(* CoDeSys 2.3.9.62 project: PackML_StateModel_Example_v2-3.pro *)
(* Libraries: STANDARD.LIB 5.6.98 13:03:02 *)

(* Global variable list: Global_Variables *)
VAR_GLOBAL
(* -------------INPUTS-------------------*)
	I_Btn_Reset			(*AT %I* *)		:BOOL;	(*Reset button*)
	I_Btn_Start			(* AT %I* *)	:BOOL;	(*Start button*)
	I_Btn_Stop			(* AT %I* *)	:BOOL;	(*Stop button*)
	I_EStopClear 		(* AT %I* *)	:BOOL :=TRUE;	(*EStop is cleared*)
	I_CoversClosed 		(* AT %I* *)	:BOOL :=TRUE;	(*Covers are completely closed*)

(* -------------OUTPUTS-------------------*)
	O_LightON_up 		(* AT %Q* *)	:BOOL;	(*Light ON - Up*)
	O_LightON_low 		(* AT %Q* *)	:BOOL;	(*Light ON - Lower*)
	OuLight_up 			(* AT %Q* *)	:INT;	(*Light Analog - Up*)
	OuLight_low 		(* AT %Q* *)	:INT;	(*Light Analog - Lower*)
	O_Light_Start 		(* AT %Q* *)	:BOOL;	(*Light Button Start*)
	O_Light_Stop 		(* AT %Q* *)	:BOOL;	(*Light Button Stop*)
	O_Light_Warning 		(* AT %Q* *):BOOL;	(*Light Button Warning*)
	O_Light_Error 		(* AT %Q* *)	:BOOL;	(*Light Button Error*)
	O_RelayStop 			(* AT %Q* *):BOOL;	(*Relay out : Stop*)
	O_RelayEStop			(* AT %Q* *):BOOL;	(*Relay out : EStop*)
	O_RelayEnableLED_Pwr_Along	(* AT %Q* *):BOOL;	(*Relay out : Enable LED power along belt*)

	bReset_System		: BOOL;			(*System reset*)
	bReset_System_Long	: BOOL;			(*System reset - Long*)
	bReqShutdown		: BOOL;			(*Request shutdown*)
	bDisplayOn			: BOOL;			(*Display on*)

(* -------------HMI INPUTS (from HMI to PLC) -------------------*)
	HMI_wControlWord	: WORD;			(*Control bits: 0=*)
	HMI_uModeReq		: UINT :=5;		(*Mode request. DEFAULT:PRODUCTION1*)

(* -------------HMI OUTPUTS (from PLC to HMI) -------------------*)
	PLC_wStatusWord		: WORD;			(*Status bits: 0=*)
	PLC_uModeCurrent	: UINT;			(*Current Mode*)
	PLC_uStateCurrent	: UINT;			(*Current State*)
	fAngle1				: REAL := 50;	(*Process: Angle1*)
	fAngle2				: REAL := 90;	(*Process: Angle2*)


(*-----------------------FUNCTION BLOCKS----------------*)
	fbStateModel		: FB_PackMLStateModel_ST;	(*FB for executing PackML state model*)

(*-----------------------OTHER GLOBAL VARS ----------------*)
	uCounterPosCurr_SIMU	: UDINT;	(*Current Counter position*)

END_VAR

(*------------------------- PERSISTENT VARIABLES --------------------------------*)
VAR_GLOBAL PERSISTENT

END_VAR

(*------------------------- CONSTANT VARIABLES --------------------------------*)
VAR_GLOBAL CONSTANT
(*-----------------------Setup Constants----------------------------*)
	bSIMU			: BOOL 	:= TRUE;	(*In simulation mode*)

(*-----------------------TIME Constants----------------------------*)
	TRESET_SYSTEM	: TIME := T#3s;		(*Delay for System Reset*)
	TRESET_LONG		: TIME := T#10s;	(*Delay for Long Reset*)

END_VAR

(* Data type *)
TYPE E_Mode :
(*UserModes: Modes for different production states*)
(
	eMode_undefined := 0,
	eMode_Automatic :=1,
	eMode_Manual :=3,
	eMode_Production1 :=5,
	eMode_Production2 :=6
);
END_TYPE

(* Data type *)
TYPE E_ModeProc :
(*Procedural control modes. Can be changed in any state*)
(
	eModeProc_undefined := 0,
	eModeProc_Automatic :=1,
	eModeProc_SemiAutomatic :=2,
	eModeProc_Manual :=3
);
END_TYPE

(* Data type *)
TYPE E_PackMLState :
(*PackML States*)
(
	eSt_Aborting :=0,
	eSt_Aborted,
	eSt_Clearing,
	eSt_Stopped,
	eSt_Stopping,
	eSt_Resetting,
	eSt_Idle,
	eSt_Starting,
	eSt_Execute,
	eSt_Suspending,
	eSt_Suspended,
	eSt_Unsuspending,
	eSt_Holding,
	eSt_Held,
	eSt_UnHolding,
	eSt_Completing,
	eSt_Completed
);
END_TYPE

(* POU Programs/PRG_Application, ST *)
PROGRAM PRG_Application
VAR
	bInitDone	: BOOL;
END_VAR
(*Application specific program routine.*)
(* It can utilise the same main state model and modes also internally, and filtter
its execution conditions according that information. Alternative option is to call
this program from Main, but only when certain conditions are met. Then special care 
should be taken what the outputs are when it is NOT called!.*)


(*Initialisation procedures*)
IF NOT bInitDone THEN
	(*TODO: Do some init actions*)
	bInitDone:=TRUE;
END_IF;

(*Mode and state analysis*)
(*Execution mode*)
IF bSIMU THEN
	PRG_SIMU();
END_IF;


IF (fbStateModel.eState >= eSt_Stopped) THEN
	(*State is equal or above Stopped*)			(*TODO: Remove/Replace this row with desired actions*)
	CASE fbStateModel.eMode OF
		(*MODE: MANUAL*)
		eMode_Manual:
			(*TODO: Do some actions in manual mode*)
			(*E.g. calling some other PRG or FB implementing manual operations*)
			;									(*TODO: Remove/Replace this row with desired actions*)

		(*MODE: AUTOMATIC*)
		eMode_Automatic:
			(*TODO: Do some actions in automatic mode*)
			(*E.g. calling some other PRG or FB implementing automatic operations*)
			;									(*TODO: Remove/Replace this row with desired actions*)
		ELSE	(*Error*)
			; (*TODO*)
	END_CASE;
END_IF;


(*Enable LED powers*)
O_RelayEnableLED_Pwr_Along := (fbStateModel.eState >= eSt_Stopped);	(*TODO: Remove/Replace this row with desired actions*)


(*Clear LED output values in case 'low' states *)
IF (fbStateModel.eState <= eSt_Clearing) THEN
	(*TODO: Actions for clearing states *)
	(*UP*)
	O_LightON_up := FALSE;				(*TODO: Remove/Replace this row with desired actions*)
	OuLight_up := 0;					(*TODO: Change...*)
	(*Low*)
	O_LightON_low := FALSE;				(*TODO: Change...*)
	OuLight_low := 0;
END_IF;
END_PROGRAM

(* POU Programs/PRG_SIMU, ST *)
PROGRAM PRG_SIMU
VAR
	c	: INT;
END_VAR
(*This just simulator part, when program is used in simulated environment*)
IF fbStateModel.eState = eSt_Clearing THEN
uCounterPosCurr_SIMU := 0;
END_IF;

IF (fbStateModel.eState > eSt_Idle) AND (fbStateModel.eState < eSt_Completed) AND
		NOT ((fbStateModel.eState = eSt_Held) OR (fbStateModel.eState = eSt_Suspended)) THEN
	c:=c+1;
	IF c >= 5 THEN
		uCounterPosCurr_SIMU := uCounterPosCurr_SIMU + 1;
		c:=0;
	END_IF;
END_IF;
END_PROGRAM

(* POU Programs/PRG_Blinking, ST *)
PROGRAM PRG_Blinking
(*Avustavia laskentaoperaatioita
- vilkutussignaalit
Author: Niko Siltala, niko.siltala@tut.fi, Tampere University of Technology / MEI
Date: 2016-12-12
Version: 1.0
*)
VAR_OUTPUT
	bSign4Hz:BOOL;					(*4 Hz (240krt/min) taajudella vaihteleva signaali*)
	bSign2Hz:BOOL;					(*2 Hz (120krt/min) taajudella vaihteleva signaali*)
	bSign1Hz:BOOL;					(*1 Hz (60krt/min) taajudella vaihteleva signaali*)
	bSign0_5Hz:BOOL;				(*0,5 Hz (30krt/min) taajudella vaihteleva signaali*)
END_VAR
VAR
	bInitDone	: BOOL	:=FALSE;	(*Ohjelman initialisointi*)
	TP_Delay:TP;				(*Nopein taajuus / 2 tuottaja*)
	bBaseHz:BOOL:=FALSE;		(*Nopein taajuus/2*)
	iBaseHz:UINT:=4;				(*Base taajuus (Hz)*)
	(*RTRIG_BASE: R_TRIG;		(*Base signaali nousee*)*)
	RTRIG_2Hz_Sign : R_TRIG;		(*2Hz signaalin generointi*)
	RTRIG_1Hz_Sign : R_TRIG;		(*1Hz signaalin generointi*)
	RTRIG_0_5Hz_Sign : R_TRIG;	(*0,5Hz signaalin generointi*)
	tBaseTaajuus:TIME;			(*Base vilkutuksen timerin arvo. f/2*)
	fPLC_CYCLE_TIME: LREAL;	(*PLC:n cycli aika. Sekunttia*)

END_VAR
(*Ohjelman initialisoinnit - Suoritetaan vain kertaalleen*)
IF NOT bInitDone THEN
	(*fPLC_CYCLE_TIME := UDINT_TO_LREAL(SystemTaskInfoArr[1].cycleTime) / 10E6; (*[s]*)*)
	fPLC_Cycle_Time := 1;	(*[s]*)
	(*Base Vilkkusignaalien tuottaminen*)
	(* 250ms - 1* cykliaika(20ms)*)
	tBaseTaajuus := LREAL_TO_TIME( ( (1/ UINT_TO_LREAL(iBaseHz) / 2 ) - 1 * fPLC_CYCLE_TIME ) * 1000);
	bInitDone := TRUE;
END_IF;

(*Base signaalin genrointi*)
TP_Delay(IN:=NOT TP_Delay.Q , PT:=tBaseTaajuus);
IF NOT TP_Delay.Q THEN
	bBaseHz := NOT bBaseHz;
	bSign4Hz:= bBaseHz;
END_IF;

(*2Hz signaalin genrointi*)
RTRIG_2Hz_Sign(CLK:=bSign4Hz);
IF RTRIG_2Hz_Sign.Q THEN
	bSign2Hz:=NOT bSign2Hz;
END_IF;

(*1Hz signaalin genrointi*)
RTRIG_1Hz_Sign(CLK:=bSign2Hz);
IF RTRIG_1Hz_Sign.Q THEN
	bSign1Hz:=NOT bSign1Hz;
END_IF;

(*0,5 Hz signaalin generointi*)
RTRIG_0_5Hz_Sign(CLK:=bSign1Hz);
IF (RTRIG_0_5Hz_Sign.Q) THEN
	bSign0_5Hz:= NOT bSign0_5Hz;
END_IF;
END_PROGRAM

(* POU Programs/PRG_Initialisation, SFC *)
PROGRAM PRG_Initialisation
(*Example program to demonstrate imagenary Initialisation and Homing process*)
VAR_INPUT
	bReset		: BOOL;	(*Performs reset*)
END_VAR
VAR_OUTPUT
	bInitDone	: BOOL;	(*Initialisation is completed*)
END_VAR
VAR
	SFCReset 	: BOOL;	(*Resets the execution of SFC to init once this SFCFlag is set true *)
END_VAR
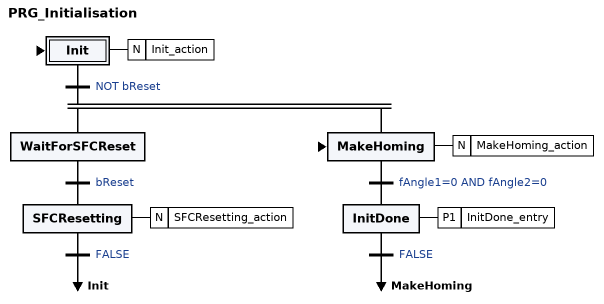
INITIAL_STEP Init:
	Init_action(N);
END_STEP
TRANSITION FROM Init TO (WaitForSFCReset, MakeHoming) := NOT bReset;
END_TRANSITION
STEP WaitForSFCReset:
END_STEP
TRANSITION FROM WaitForSFCReset TO SFCResetting := bReset;
END_TRANSITION
STEP SFCResetting:
	SFCResetting_action(N);
END_STEP
TRANSITION FROM SFCResetting TO Init := FALSE;
END_TRANSITION
STEP MakeHoming:
	MakeHoming_action(N);
END_STEP
TRANSITION FROM MakeHoming TO InitDone := fAngle1=0 AND fAngle2=0;
END_TRANSITION
STEP InitDone:
	InitDone_entry(P1);
END_STEP
TRANSITION FROM InitDone TO MakeHoming := FALSE;
END_TRANSITION

ACTION Init_action:
SFCReset := FALSE;
bReset	:= FALSE;
END_ACTION

ACTION SFCResetting_action:
SFCReset := TRUE;
END_ACTION

ACTION MakeHoming_action:
bInitDone := FALSE;
(*Return pointer1 to home. CCW rotation*)
fAngle1 := fAngle1 - 0.5;
IF fAngle1 <= 0 THEN
	fAngle1 := 0;
END_IF;

(*Return pointer2 to home. CCW rotation*)
IF fAngle2 <> 0 THEN
	IF fAngle2 < 0 THEN
		fAngle2 := fAngle2 + 360;
	END_IF;
	fAngle2 := fAngle2 - 0.5;
	IF fAngle2 <= 0 THEN
		fAngle2 := 0;
	END_IF;
END_IF;
END_ACTION

ACTION InitDone_entry:
bInitDone := TRUE;
END_ACTION
END_PROGRAM

(* POU PRG_MAIN, ST *)
PROGRAM PRG_MAIN
VAR
	TON_Reset_Long		: TON;
	TON_Reset_System	: TON;
	tonStarting			: TON;
	bBlink				: BOOL;	(*1s blinking for CodeSys Simulation*)
	c					: INT;	(*Support variable for blinking*)
	fbProcess3		: FB_Process3; (*FB Instance representing Process 3 *)
END_VAR
(* ****** Section 1: Initialisations and default values. Initial conditions for variables on every PLC cycle*)
fbStateModel.bSC := FALSE;
fbProcess3.packML_State := fbStateModel.eState;
fbProcess3.packML_Mode := fbStateModel.eMode;

PRG_MAIN_SAMPLE();

IF bSIMU THEN
	(*TODO set counter source*)
	;
END_IF;

(*System resets*)
TON_Reset_System(IN:=I_Btn_Reset,
		PT:=TRESET_SYSTEM ,
		Q=> , ET=> );		(*Simple Reset actions should happen after this*)
TON_Reset_Long(IN:=I_Btn_Reset,
		PT:=TRESET_LONG ,
		Q=>bReset_System_Long , ET=> );	(*Complete Reset actions should happen after this*)
bReset_System := TON_Reset_System.Q;

(* ****** Section 2: Grouping PackML states for calling Programs or FB instances.
This is to avoid repetition inside case structure in Section 3. With IF clause setting lower (and upper) state limits we can filter out the states when we want to call 
specific programs. The order of states is defined in Tab:Data types > E_PackMLState. eSt_Aborting is lowest and eSt_Completed is highest.
Here we filter calling programs, only when we are in higher states than Stopped. Inside IF there is again CASE which process each Control Mode separately.*)
(*Execution part. Making calls for program if we are on states above Stopped*)
IF (fbStateModel.eState > eSt_Stopped) THEN
	(*State is equal or above Stopped*)			(*TODO: Remove/Replace this row with desired actions*)
	CASE fbStateModel.eMode OF
		(*MODE: MANUAL*)
		eMode_Manual:
			(*TODO: Do some actions in manual mode*)
			(*E.g. calling some other PRG or FB implementing manual operations*)
			;									(*TODO: Remove/Replace this row with desired actions*)

		(*MODE: PRODUCTION1*)
		eMode_Production1:
			(*TODO: Do some actions in production1 mode*)
			(*E.g. calling some other PRG or FB implementing automatic operations*)
			PRG_Production1();					(*TODO: Remove/Replace this row with desired actions*)
			;									(*TODO: Remove/Replace this row with desired actions*)
			(*Calling Process 3*)
			fbProcess3(
				bReset:= FALSE);

		(*MODE: PRODUCTION2*)
		eMode_Production2:
			(*TODO: Do some actions in production2 mode*)
			(*E.g. calling some other PRG or FB implementing automatic operations*)
			PRG_Production1();					(*TODO: Remove/Replace this row with desired actions*)
			PRG_Production2();					(*TODO: Remove/Replace this row with desired actions*)
		ELSE	(*Error*)
			; (*TODO*)
	END_CASE;
END_IF;

(* ****** Section 3: Actions in your program without considering the Control Mode. I.e. actions are performed same way indenpendent on
current Control Mode selection.*)
(*PackML state actions which are Mode independent*)
CASE fbStateModel.eState OF
eSt_Aborting:
	(*Make here possible power off or braking procedures. The same action could be called from multiple places.*)
	actAborting;
	PRG_Initialisation(bReset := TRUE);
	fbProcess3(
		bReset:= TRUE);
	fbStateModel.bSC := TRUE;		(*TODO: Remove/Replace this row with desired actions*)
eSt_Clearing:
	(*Make here clearing and reseting actions*)
	PRG_Initialisation(bReset := FALSE);
	fbProcess3(
		bReset:= FALSE);
	uCounterPosCurr_SIMU:=0;		(*TODO: Remove/Replace this row. It is for demo actions.*)
	fbStateModel.bSC := TRUE;		(*TODO: Remove/Replace this row with desired actions*)
eSt_Resetting:
	fbStateModel.bSC := TRUE;		(*TODO: Remove/Replace this row with desired actions*)
eSt_Holding:
	fbStateModel.bSC := TRUE;		(*TODO: Remove/Replace this row with desired actions*)
eSt_UnHolding:
	fbStateModel.bSC := TRUE;		(*TODO: Remove/Replace this row with desired actions*)
eSt_Suspending:
	fbStateModel.bSC := TRUE;		(*TODO: Remove/Replace this row with desired actions*)
eSt_Unsuspending:
	fbStateModel.bSC := TRUE;		(*TODO: Remove/Replace this row with desired actions*)
END_CASE;

(* ****** Section 4: Actions in your program which are Control Mode specific. Two nested case structures where outer one selects the
control mode and inner the PackML state. In order to avoid conflicts, it would be better to process each PackML state either in Section 2 
or Section 3, but not in both. *)
(*PackML state actions related to User/Production mode *)
CASE fbStateModel.eMode OF
(*MODE: MANUAL*)
eMode_Manual:
	(* ****** Section 3.1: PackML state based processing actions when Control Mode is Manual.*)
	CASE fbStateModel.eState OF
	eSt_Idle:
		fbStateModel.bAck_Completed := FALSE;		(*TODO: Remove/Replace this row with desired actions*)
	eSt_Starting:
		fbStateModel.bSC := TRUE;		(*TODO: Remove/Replace this row with desired actions*)
	eSt_Completing:
		fbStateModel.bSC := TRUE;		(*TODO: Remove/Replace this row with desired actions*)
	eSt_Completed:
		fbStateModel.bAck_Completed := TRUE;		(*TODO: Remove/Replace this row with desired actions*)
	eSt_Stopping:
		fbStateModel.bSC := TRUE;		(*TODO: Remove/Replace this row with desired actions*)
	END_CASE;

(*MODE: PRODUCTION1*)
eMode_Production1:
	(* ****** Section 3.2: PackML state based processing actions when Control Mode is Production 1.*)
	CASE fbStateModel.eState OF
	eSt_Idle:
		fbStateModel.bAck_Completed := FALSE;			(*TODO: Remove/Replace this row with desired actions*)
		tonStarting(IN:=FALSE , PT:= , Q=> , ET=> );	(*TODO: Remove/Replace this row. It is for demo actions.*)
	eSt_Starting:
		tonStarting(IN:=TRUE , PT:=T#2s , Q=> , ET=> );	(*TODO: Remove/Replace this row. It is for demo actions.*)
		PRG_Initialisation(bInitDone=> );				(*TODO: Remove/Replace this row with desired actions*)
		fbStateModel.bSC := tonStarting.Q AND PRG_Initialisation.bInitDone AND fbProcess3.bInitDone;		(*TODO: Remove/Replace this row with desired actions*)
	eSt_Completing:
		fbStateModel.bSC := PRG_Production1.bStopOK;			(*TODO: Remove/Replace this row with desired actions*)
	eSt_Completed:
		;
		(*fbStateModel.bAck_Completed:= I_Btn_Start;*)
	eSt_Stopping:
		(*fbStateModel.bSC := TRUE;		*)(*TODO: Remove/Replace this row with desired actions*)
		fbStateModel.bSC := NOT PRG_Initialisation.bInitDone OR (PRG_Production1.bStopOK AND fbProcess3.bStopOK);	(*TODO: Remove/Replace this row with desired actions*)
	END_CASE;

(*MODE: PRODUCTION2*)
eMode_Production2:
	CASE fbStateModel.eState OF
	eSt_Idle:
		fbStateModel.bAck_Completed := FALSE;			(*TODO: Remove/Replace this row with desired actions*)
		tonStarting(IN:=FALSE , PT:= , Q=> , ET=> );	(*TODO: Remove/Replace this row. It is for demo actions.*)
	eSt_Starting:
		tonStarting(IN:=TRUE , PT:=T#0s , Q=> , ET=> );	(*TODO: Remove/Replace this row. It is for demo actions.*)
		PRG_Initialisation(bInitDone=> );				(*TODO: Remove/Replace this row with desired actions*)
		fbStateModel.bSC := tonStarting.Q AND PRG_Initialisation.bInitDone;		(*TODO: Remove/Replace this row with desired actions*)
	eSt_Completing:
		fbStateModel.bSC := (PRG_Production1.bStopOK AND PRG_Production2.bStopOK);	(*TODO: Remove/Replace this row with desired actions*)
	eSt_Completed:
		;
		(*fbStateModel.bAck_Completed:= I_Btn_Start;*)
	eSt_Stopping:
		fbStateModel.bSC := NOT PRG_Initialisation.bInitDone OR (PRG_Production1.bStopOK AND PRG_Production2.bStopOK);	(*TODO: Remove/Replace this row with desired actions*)
	END_CASE;

(*MODE: UNKNOWN*)
ELSE	(*This is an Error branch.*)
	; (*TODO: Make implementation*)
END_CASE;

(* ****** Section 5: Calling the fbStateModel instance.
Here the instance of state model is called and all triggering inputs are set, but bSC (State Completed), which you control in your programs. This is indication that your program 
has  finished certain stage.
- Pay attention where the instance fbStateModel is defined. Do you do it in global variables or e.g. here in PRG_MAIN? Important is to use the same instance in all places, so that
machine state is unique and shared. Remember, if you have multiple definitions, the PRG_MAIN "hides" the global one, and might lead to problems elswhere, when you think you 
are using the same instance, but actually are not. 
- In case you are using the PackML visualisation (VC_PackMLStates), make sure you connect its placeholder to the very same PackML FB instance.
- The Mask for wIgnoreState is created as following. I use binary base for the value(2#). The lowest bit in the mask corresponds the  eSt_Aborting in E_PackMLState.
The next is eSt_Aborted, and so on. Specific state is ignored and jumped over when it is masked out i.e. ignored by having 1 in that position. Note that implementation allows 
this only for selected states. See FB_PackMLStateModel_ST code for further details.*)
(*Calling & Updating the state model*)
(*TODO: Evaluate and change all input conditions according your application needs*)
fbStateModel(
	bResetFB:= bReset_System_Long,
	eModeReq:= HMI_uModeReq,
	wIgnoreState := 2#000000,		(*TODO: Which states should be ignodered. Default: 2#100000*)
	bSC:= ,			(*Must NOT be assigned ANY variable, because fb input is directly assigned above!!!*)
	bAbort:= bReset_System OR bReqShutdown OR NOT (I_CoversClosed AND I_EStopClear),
	bClear:= I_Btn_Reset,
	bReset:= I_Btn_Start,
	bStart:= (I_Btn_Start OR HMI_wControlWord.1) AND I_EStopClear,
	bHold:= HMI_wControlWord.3,
	bUn_Hold:= I_Btn_Reset OR HMI_wControlWord.5 OR HMI_wControlWord.7,
	bSuspend:= HMI_wControlWord.4,
	bUn_Suspend:= I_Btn_Reset OR HMI_wControlWord.6 OR HMI_wControlWord.7,
	bStop:= I_Btn_Stop OR HMI_wControlWord.2,
	bComplete:= ,
	bAck_Completed:= ,
	eMode=> PLC_uModeCurrent,
	eState=> PLC_uStateCurrent);

(* ****** Section 6: Here we update all outputs according the current state of our PackML model. This allows us to process the in single location.
The control of outputs is bind to state, not e.g. to inputs. The inputs are the one driving the PackML model forward. Again CASE structure can be used.*)
(*Call for HMI and UI update*)
HMI_and_UI_Update;
END_PROGRAM
ACTION actAborting:
(*Add here Aborting related actions*)
;
END_ACTION
ACTION HMI_and_UI_Update:
(*HMI Update*)
(*Calling blinking sub-program*)
PRG_Blinking (bSign4Hz=> , bSign2Hz=> , bSign1Hz=> , bSign0_5Hz=> );

(*Codesys simulation 1Hz blinking*)
c:= c + 1;
IF c > 1 THEN
	c:=0;
END_IF;
bBlink := (c=0);	(*Blink is true if c=0*)

(*Init values*)
O_Light_Stop := FALSE;	(*TODO: Change initial values according your app needs*)
O_Light_Warning:=FALSE;	(*TODO: Change initial values according your app needs*)
O_Light_Error:=FALSE;	(*TODO: Change initial values according your app needs*)

(*TODO: Change values according range of states *)
(*Start light*)
O_Light_Start :=  (fbStateModel.eState >= eSt_Resetting) AND (fbStateModel.eState < eSt_Completed);

(*TODO: Change output values according states *)
CASE fbStateModel.eState OF
eSt_Aborting, eSt_Aborted:
	O_Light_Stop := bBlink;	(*TODO: Change initial values according your app needs*)
	O_RelayStop := FALSE;					(*TODO: Change initial values according your app needs*)
	O_RelayEStop := FALSE;					(*TODO: Change initial values according your app needs*)
eSt_Clearing:
	O_Light_Stop := bBlink; 					(*TODO: Change initial values according your app needs*)
eSt_Stopping:
	O_Light_Stop := bBlink;					(*TODO: Change initial values according your app needs*)
	O_RelayStop := FALSE;					(*TODO: Change ...*)
eSt_Stopped, eSt_Completed:
	O_Light_Stop := TRUE;					(*TODO: Change initial values according your app needs*)
	O_RelayStop := FALSE;					(*TODO: Change ...*)
eSt_Starting:
	O_Light_Start := bBlink;					(*TODO: Change ...*)
	O_RelayStop := TRUE;						(*TODO: Change ...*)
	O_RelayEStop := TRUE;					(*TODO: Change ...*)
END_CASE;
END_ACTION

(* POU Programs/FB_Process3, SFC *)
FUNCTION_BLOCK FB_Process3
VAR_INPUT
	bReset		: BOOL;	(*Reset Request*)
	packML_State	: E_PackMLState;
	packML_Mode	: E_Mode;
END_VAR
VAR_OUTPUT
	bInitDone		: BOOL; 	(*Initialisation completed*)
	bStopOK		: BOOL;	(*Stopping OK*)
END_VAR
VAR
	iProcessCount	: INT := 0;	(*Counter for demonstrating process*)
	bLocalReset	: BOOL;	(*Performs local reset*)
	SFCReset 	: BOOL;	(*Resets the execution of SFC to init once this SFCFlag is set true *)
END_VAR
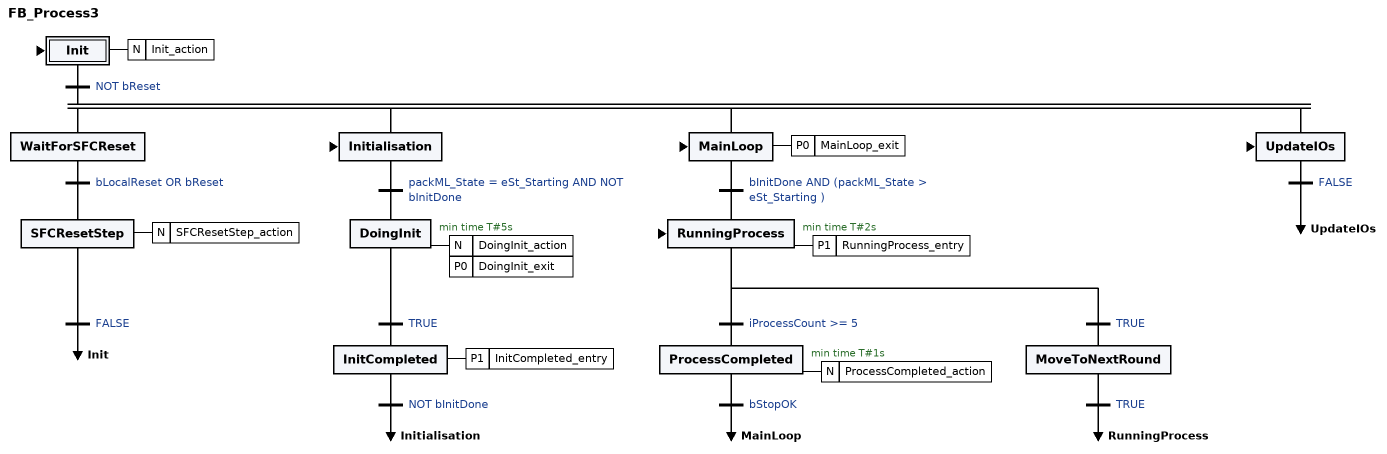
INITIAL_STEP Init:
	Init_action(N);
END_STEP
TRANSITION FROM Init TO (WaitForSFCReset, Initialisation, MainLoop, UpdateIOs) := NOT bReset;
END_TRANSITION
STEP WaitForSFCReset:
END_STEP
TRANSITION FROM WaitForSFCReset TO SFCResetStep := bLocalReset OR bReset;
END_TRANSITION
STEP SFCResetStep:
	SFCResetStep_action(N);
END_STEP
TRANSITION FROM SFCResetStep TO Init := FALSE;
END_TRANSITION
STEP Initialisation:
END_STEP
TRANSITION FROM Initialisation TO DoingInit := packML_State = eSt_Starting AND NOT bInitDone;
END_TRANSITION
STEP DoingInit: (* min time T#5s *)
	DoingInit_action(N);
	DoingInit_exit(P0);
END_STEP
TRANSITION FROM DoingInit TO InitCompleted := TRUE;
END_TRANSITION
STEP InitCompleted:
	InitCompleted_entry(P1);
END_STEP
TRANSITION FROM InitCompleted TO Initialisation := NOT bInitDone;
END_TRANSITION
STEP MainLoop:
	MainLoop_exit(P0);
END_STEP
TRANSITION FROM MainLoop TO RunningProcess := bInitDone AND (packML_State > eSt_Starting );
END_TRANSITION
STEP RunningProcess: (* min time T#2s *)
	RunningProcess_entry(P1);
END_STEP
TRANSITION FROM RunningProcess TO ProcessCompleted := iProcessCount >= 5;
END_TRANSITION
TRANSITION FROM RunningProcess TO MoveToNextRound := TRUE;
END_TRANSITION
STEP ProcessCompleted: (* min time T#1s *)
	ProcessCompleted_action(N);
END_STEP
TRANSITION FROM ProcessCompleted TO MainLoop := bStopOK;
END_TRANSITION
STEP MoveToNextRound:
END_STEP
TRANSITION FROM MoveToNextRound TO RunningProcess := TRUE;
END_TRANSITION
STEP UpdateIOs:
END_STEP
TRANSITION FROM UpdateIOs TO UpdateIOs := FALSE;
END_TRANSITION

ACTION Init_action:
SFCReset := FALSE;
bLocalReset	:= FALSE;
bInitDone := FALSE;
END_ACTION

ACTION SFCResetStep_action:
SFCReset := TRUE;
END_ACTION

ACTION DoingInit_action:
iProcessCount := 0;
END_ACTION

ACTION DoingInit_exit:
bStopOK := TRUE;
END_ACTION

ACTION InitCompleted_entry:
bInitDone := TRUE;
END_ACTION

ACTION MainLoop_exit:
bStopOK  := FALSE;
END_ACTION

ACTION RunningProcess_entry:
iProcessCount := iProcessCount + 1;
END_ACTION

ACTION ProcessCompleted_action:
bStopOK  := TRUE;
iProcessCount := 0;
END_ACTION
END_FUNCTION_BLOCK

(* POU Examples/PRG_MAIN_SAMPLE, ST *)
PROGRAM PRG_MAIN_SAMPLE
VAR
(*	fbStateModel		: FB_PackMLStateModel_ST;	(*FB for executing PackML state model*)		*)
	bBlink				: BOOL;	(*1s blinkg for CodeSys Simulation*)
	c					: INT;	(*Support variable for blinking*)
END_VAR
(* ****** Section 1: Initialisations and default values. Initial conditions for variables on every PLC cycle*)
fbStateModel.bSC := FALSE;

(* ****** Section 2: Grouping PackML states for calling Programs or FB instances.
This is to avoid repetition inside case structure in Section 4. With IF clause setting lower (and upper) state limits we can filter out the states when we 
want to call specific programs. The order of states is defined in Tab:Data types > E_PackMLState. eSt_Aborting is the lowest and eSt_Completed is 
the highest. Here we filter out calling of the programs - we call them only when we are in higher states than Stopped. Inside IF there is again CASE 
which process each Control Mode separately.*)
(*Execution part. Making calls for program if we are on states above Stopped*)
IF (fbStateModel.eState > eSt_Stopped) THEN
	CASE fbStateModel.eMode OF
		(*MODE: MANUAL*)
		eMode_Manual:
			;
		(*MODE: AUTOMATIC*)
		eMode_Automatic:
			;
	END_CASE;
END_IF;

(* ****** Section 3: Actions in your program without considering the Control Mode. I.e. actions are performed same way indenpendent on
current Control Mode selection.*)
(*Mode independent state actions*)
CASE fbStateModel.eState OF
eSt_Aborting:
	(* One can make specific actions in case of specific Mode-State combination.
	   One can also consider to call a specific program when in specific Mode-State combination*)
	actAborting;
	fbStateModel.bSC := TRUE;		(*TODO: Remove/Replace this row with desired actions*)
eSt_Clearing:
	fbStateModel.bSC := TRUE;		(*TODO: Remove/Replace this row with desired actions*)
eSt_Stopping:
	fbStateModel.bSC := TRUE;		(*TODO: Remove/Replace this row with desired actions*)
eSt_Resetting:
	fbStateModel.bSC := TRUE;		(*TODO: Remove/Replace this row with desired actions*)
eSt_Holding:
	fbStateModel.bSC := TRUE;		(*TODO: Remove/Replace this row with desired actions*)
eSt_UnHolding:
	fbStateModel.bSC := TRUE;		(*TODO: Remove/Replace this row with desired actions*)
eSt_Suspending:
	fbStateModel.bSC := TRUE;		(*TODO: Remove/Replace this row with desired actions*)
eSt_Unsuspending:
	fbStateModel.bSC := TRUE;		(*TODO: Remove/Replace this row with desired actions*)
END_CASE;

(* ****** Section 4: Actions in your program which are Control Mode specific. Two nested case structures where outer one selects the
control mode and inner the PackML state. In order to avoid conflicts, it would be better to process each PackML state either in Section 3 
or Section 4, but not in both. *)
(*Execution mode related state actions*)
CASE fbStateModel.eMode OF
(*MODE: MANUAL*)
eMode_Manual:
	(* ****** Section 4.1: PackML state based processing actions when Control Mode is Manual.*)
	CASE fbStateModel.eState OF
	eSt_Idle:
		fbStateModel.bAck_Completed := FALSE;		(*TODO: Remove/Replace this row with desired actions*)
	eSt_Starting:
		fbStateModel.bSC := TRUE;					(*TODO: Remove/Replace this row with desired actions*)
	eSt_Completing:
		fbStateModel.bSC := TRUE;					(*TODO: Remove/Replace this row with desired actions*)
	eSt_Completed:
		fbStateModel.bAck_Completed := TRUE;		(*TODO: Remove/Replace this row with desired actions*)
	END_CASE;

(*MODE: AUTOMATIC*)
eMode_Automatic:
	(* ****** Section 4.2: PackML state based processing actions when Control Mode is Automatic.*)
	CASE fbStateModel.eState OF
	eSt_Idle:
		fbStateModel.bAck_Completed := FALSE;		(*TODO: Remove/Replace this row with desired actions*)
	eSt_Starting:
		fbStateModel.bSC := TRUE;					(*TODO: Remove/Replace this row with desired actions*)
	eSt_Completing:
		fbStateModel.bSC := TRUE;					(*TODO: Remove/Replace this row with desired actions*)
	eSt_Completed:
		;
		(*fbStateModel.bAck_Completed:= TRUE;*)
	END_CASE;

(*MODE: UNKNOWN*)
ELSE	(*This is an Error branch.*)
	; (*TODO: Make implementation*)
END_CASE;

(* ****** Section 5: Calling the fbStateModel instance.
Here the instance of state model is called and all triggering inputs are set, but bSC (State Completed), which you control in your programs. 
This is indication that your program has  finished certain stage.
- Pay attention where the instance fbStateModel is defined. Do you do it in global variables or e.g. here in PRG_MAIN? Important is to use the 
same instance in all places, so that machine state is unique and shared. Remember, if you have multiple definitions, the PRG_MAIN "hides" 
the global one, and might lead to problems elswhere, when you think you are using the same instance, but actually are not. 
- In case you are using the PackML visualisation (VC_PackMLStates), make sure you connect its placeholder to the very same PackML FB instance.
- The Mask for wIgnoreState is created as following. I use binary base for the value(2#). The lowest bit in the mask corresponds the eSt_Aborting
 in E_PackMLState. The next is eSt_Aborted, and so on. Specific state is ignored and jumped over when it is masked out i.e. ignored by having 1 
in that position. Note that implementation allows this only for selected states. See FB_PackMLStateModel_ST code for further details.*)
(*Calling & Updating the state model*)
(*TODO: Evaluate and change all input conditions according your application needs*)
fbStateModel(
	bResetFB:= ,
	eModeReq:= ,
	wIgnoreState := 2#000000,		(*TODO: Which states should be ignodered. Default: 2#000000 or 2#100000*)
	bSC:= ,		(*Must NOT be assigned ANY variable, because fb input is directly assigned above by your programs!!!*)
	bAbort:= ,
	bClear:= ,
	bReset:= ,
	bStart:= ,
	bHold:= ,
	bUn_Hold:= ,
	bSuspend:= ,
	bUn_Suspend:= ,
	bStop:= ,
	bComplete:= ,
	bAck_Completed:= ,
	eMode=> ,
	eState=> );

(* ****** Section 6: Here we update all outputs according the current state of our PackML model. This allows us to process the in single location.
The control of outputs is bind to state, not e.g. to inputs. The inputs are the one driving the PackML model forward. Again CASE structure can be used.*)
(*Call for HMI and UI update*)
HMI_and_UI_Update;
END_PROGRAM
ACTION actAborting:
(*You can add here Aborting related actions as one central collection.
This action can be called from multiple places, in case needed, 
but is part of program*)
;
END_ACTION
ACTION HMI_and_UI_Update:
(*HMI Update*)
(*Calling blinking sub-program*)
(*PRG_Blinking (bSign4Hz=> , bSign2Hz=> , bSign1Hz=> , bSign0_5Hz=> );*)
(*Codesys simulation 1Hz blinking*)
c:= c + 1;
IF c > 1 THEN
	c:=0;
END_IF;
bBlink := (c=0);	(*bBlink is true if c=0*)

(*Init values*)
O_Light_Stop := FALSE;	(*TODO: Change initial values according your app needs*)

(*TODO: Change values according range of states *)
(*Start light*)
(*O_Light_Start :=  (fbStateModel.eState >= eSt_Resetting) AND (fbStateModel.eState < eSt_Completed); *)

(*TODO: Change output values according states *)
CASE fbStateModel.eState OF
eSt_Aborting, eSt_Aborted:
	O_Light_Stop := bBlink;					(*TODO: Change initial values according your app needs*)
eSt_Clearing:
	O_Light_Stop := bBlink; 					(*TODO: Change initial values according your app needs*)
eSt_Stopping, eSt_Stopped, eSt_Completed:
	O_Light_Stop := TRUE;					(*TODO: Change initial values according your app needs*)
eSt_Starting:
	;
	(*O_Light_Start := bBlink;	*)				(*TODO: Change initial values according your app needs*)
END_CASE;
END_ACTION

(* POU Programs/PRG_Production1, ST *)
PROGRAM PRG_Production1
(*Example program to demonstrate imagenary Production1 process*)
VAR_INPUT
	bReset		: BOOL;	(*Performs reset*)
END_VAR
VAR_OUTPUT
	bStopOK		: BOOL;	(*Stopping OK*)
END_VAR
VAR
	iCycleCount	: INT;	(*Cycle counter*)
END_VAR
bStopOK := FALSE;

CASE fbStateModel.eState OF
eSt_Execute:		(*Actions during normal execution*)
	fAngle1 := fAngle1 + 4;
(*	IF fAngle1 >= 360 THEN
		fAngle1 := 0;
		iCycleCount := iCycleCount +1;
	END_IF;*)

eSt_Stopping, eSt_Completing :
(*What should happen during stopping*)
	IF fAngle1 <> 0 THEN
		fAngle1 := fAngle1 + 4;
	END_IF;
(*	IF fAngle1 >= 360 THEN
		fAngle1 := 0;
		iCycleCount := iCycleCount +1;
	END_IF;*)

	(*Stopping condition*)
	IF fAngle1 = 0 THEN
		bStopOK := TRUE;
	END_IF;

END_CASE;

(*Check angle overrun*)
IF fAngle1 >= 360 THEN
	fAngle1 := 0;
	iCycleCount := iCycleCount +1;
END_IF;
END_PROGRAM

(* POU Programs/PRG_Production2, ST *)
PROGRAM PRG_Production2
(*Example program to demonstrate imagenary Production2 process*)
VAR_INPUT
	bReset		: BOOL;	(*Performs reset*)
END_VAR
VAR_OUTPUT
	bStopOK		: BOOL;	(*Stopping OK*)
END_VAR
VAR
	iCycleCount	: INT;	(*Cycle counter*)
END_VAR
bStopOK := FALSE;

CASE fbStateModel.eState OF
eSt_Execute:		(*Actions during normal execution*)
	fAngle2 := fAngle2 - 3;


eSt_Stopping, eSt_Completing : (*What should happen during stopping*)
	IF fAngle2 <> 0 THEN
		fAngle2 := fAngle2 - 3;
	END_IF;
	(*Stopping condition*)
	IF (fAngle2 = 0) THEN
		bStopOK := TRUE;
	END_IF;
END_CASE;

(*Check angle overrun*)
IF fAngle2 <= -360 THEN
	fAngle2 := 0;
	iCycleCount := iCycleCount +1;
END_IF;
END_PROGRAM

(* POU FBs/FB_PackMLStateModel_ST, ST *)
FUNCTION_BLOCK FB_PackMLStateModel_ST
(*PackML State model implementation for applications.
Author: Niko Siltala, niko.siltala@tut.fi, Tampere University of Technology / MEI
Date: 2016-12-12
Version: 1.0
*)
VAR_INPUT
	bResetFB	: BOOL;		(*Resets whole FB*)
	eModeReq	: E_Mode;	(*Requested mode*)
	wIgnoreState: DWORD;	(*Ignoring states. See bit from E_PackMLState definition. Aborting = bit0*)
	bSC			: BOOL;		(*Step Completed acknoledgement*)
	bAbort		: BOOL;		(*Abortting signal = EmergencyStop*)
	bClear		: BOOL;		(*Clear signal*)
	bReset		: BOOL;		(*Reseting signal*)
	bStart		: BOOL;		(*Start signal*)
	bHold		: BOOL;		(*Hold signal*)
	bUn_Hold	: BOOL;		(*Un-Hold signal*)
	bSuspend	: BOOL;		(*Suspend signal*)
	bUn_Suspend	: BOOL;		(*Un-Suspend signal*)
	bStop		: BOOL;		(*Stop signal*)
	bComplete	: BOOL;		(*Complete signal*)
	bAck_Completed	: BOOL;	(*Acknoledgement for Complete signal*)
END_VAR
VAR_OUTPUT
	eMode	: E_Mode;		(*Current mode*)
	eState	: E_PackMLState;(*Current state*)
	strState : STRING(15);		(*State as String*)
END_VAR
VAR
	RTrig_bSC		: R_TRIG; 		(*Rising trigger for State Completed*)
	RTrig_StateChange : R_TRIG; 	(*Rising trigger for State signal*)
	bResetLocal		: BOOL:=FALSE;	(*Paikallinen Reset*)
	bInitDone		: BOOL;			(*Initialisation*)
END_VAR
IF bResetFB THEN	(*Reseting FB*)
	bInitDone := FALSE;
END_IF;

(*Initialisation*)
IF NOT bInitDone THEN
	eState:= eSt_Aborting;
	strState:='Aborting';
	bInitDone:=TRUE;
END_IF;

(*Rising triggers monitor*)
RTrig_bSC(CLK:=bSC , Q=> );

(*Abort signal interrupt*)
IF bAbort AND (eState > eSt_Clearing) THEN
	eState:=eSt_Aborting;
END_IF;

(*Stop signal interrupt*)
IF bStop AND (eState > eSt_Stopping) THEN
	eState:=eSt_Stopping;
END_IF;


(*Main case structure*)
CASE eState OF
eSt_Aborting:
	strState:='Aborting';
	IF bSC THEN
		eState:=eSt_Aborted;
	END_IF;

eSt_Aborted:
	strState:='Aborted';
	eMode:=eModeReq;	(*Change Mode allowed*)
	IF bClear AND NOT bAbort THEN
		eState:=eSt_Clearing;
	END_IF;

eSt_Clearing:
	strState:='Clearing';
	IF bAbort THEN
		eState:=eSt_Aborting;
	ELSIF bSC THEN
		eState:=eSt_Stopped;
		RTrig_StateChange(CLK:=bReset , Q=> );
	END_IF;

eSt_Stopping:
	strState:='Stopping';
	IF bSC THEN
		eState:=eSt_Stopped;
		RTrig_StateChange(CLK:=bReset , Q=> );
	END_IF;

eSt_Stopped:
	strState:='Stopped';
	eMode:=eModeReq;	(*Change Mode allowed*)
	RTrig_StateChange(CLK:=bReset , Q=> );
(*	ELSIF NOT bStop AND (RTrig_StateChange.Q OR (wIgnoreState.5 AND bStart) ) THEN*)
	IF NOT bStop THEN	(*Stop signal is not active.*)
		IF wIgnoreState.5 AND bStart THEN	(*Reset state is ignored and going directly to start *)
			eState:=eSt_Idle;
(*		ELSIF RTrig_StateChange.Q THEN 	(*Rising edge for reset*)*)
		ELSIF bReset THEN 	(*Reset*)
			eState:=eSt_Resetting;
		END_IF;
	END_IF;

eSt_Resetting:
	strState:='Resetting';
	IF bSC OR wIgnoreState.5 THEN
		eState:=eSt_Idle;
	END_IF;

eSt_Idle:
	strState:='Idle';
	eMode:=eModeReq;	(*Change Mode allowed*)
	IF bStart OR wIgnoreState.6 THEN (* IDLE state is ignoered*)
		eState:=eSt_Starting;
	END_IF;

eSt_Starting:
	strState:='Starting';
	IF bSC OR wIgnoreState.7 THEN (* STARTING state is ignoered*)
		eState:=eSt_Execute;
	END_IF;

eSt_Execute:
	strState:='Execute';
	IF bComplete THEN
		eState:=eSt_Completing;
	ELSIF bHold THEN
		eState:=eSt_Holding;
	ELSIF bSuspend THEN
		eState:=eSt_Suspending;
	END_IF;

eSt_Holding:
	strState:='Holding';
	IF bSC THEN
		eState:=eSt_Held;
	END_IF;

eSt_Held:
	strState:='Held';
	IF bUn_Hold AND NOT bHold THEN
		eState:=eSt_UnHolding;
	END_IF;

eSt_UnHolding:
	strState:='Un-Holding';
	IF bSC THEN
		eState:=eSt_Execute;
	END_IF;

eSt_Suspending:
	strState:='Suspending';
	IF bSC THEN
		eState:=eSt_Suspended;
	END_IF;

eSt_Suspended:
	strState:='Suspended';
	IF bUn_Suspend AND NOT bSuspend THEN
		eState:=eSt_Unsuspending;
	END_IF;

eSt_Unsuspending:
	strState:='Un-Suspending';
	IF bSC THEN
		eState:=eSt_Execute;
	END_IF;

eSt_Completing:
	strState:='Completing';
	IF RTrig_bSC.Q THEN
		eState:=eSt_Completed;
	END_IF;

eSt_Completed:
	strState:='Completed';
	IF bReset OR bAck_Completed THEN
		eState:=eSt_Resetting;
	END_IF;

ELSE
	(*Default error handler. Undefined state set*)
	eState:=eSt_Aborting;
END_CASE;
END_FUNCTION_BLOCK

(* POU Examples/FB_SFC_Example, SFC *)
FUNCTION_BLOCK FB_SFC_Example
VAR_INPUT
	bReset		: BOOL;	(*Reset Request*)
END_VAR
VAR_OUTPUT
END_VAR
VAR
	bLocalReset	: BOOL;	(*Performs local reset*)
	SFCReset 	: BOOL;	(*Resets the execution of SFC to init once this SFCFlag is set true *)
END_VAR
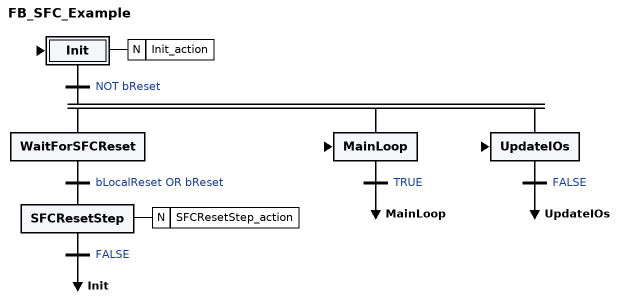
INITIAL_STEP Init:
	Init_action(N);
END_STEP
TRANSITION FROM Init TO (WaitForSFCReset, MainLoop, UpdateIOs) := NOT bReset;
END_TRANSITION
STEP WaitForSFCReset:
END_STEP
TRANSITION FROM WaitForSFCReset TO SFCResetStep := bLocalReset OR bReset;
END_TRANSITION
STEP MainLoop:
END_STEP
TRANSITION FROM MainLoop TO MainLoop := TRUE;
END_TRANSITION
STEP UpdateIOs:
END_STEP
TRANSITION FROM UpdateIOs TO UpdateIOs := FALSE;
END_TRANSITION
STEP SFCResetStep:
	SFCResetStep_action(N);
END_STEP
TRANSITION FROM SFCResetStep TO Init := FALSE;
END_TRANSITION

ACTION Init_action:
SFCReset := FALSE;
bLocalReset	:= FALSE;
END_ACTION

ACTION SFCResetStep_action:
SFCReset := TRUE;
END_ACTION
END_FUNCTION_BLOCK

(* Visualisation V_StateModelTest
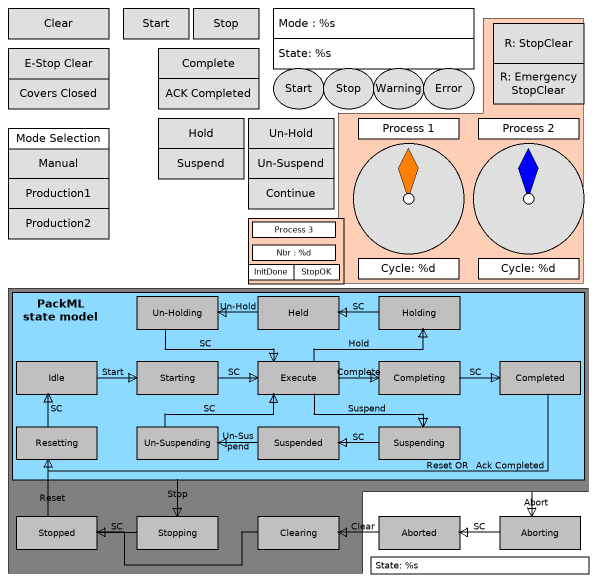
rectangle at (0,-10)-(101,21): text "Clear"; alarm colour if .I_Btn_Reset OR .HMI_wControlWord.0; taps .I_Btn_Reset
rectangle at (115,-10)-(181,21): text "Start"; alarm colour if .I_Btn_Start OR .HMI_wControlWord.1; taps .I_Btn_Start
rectangle at (185,-10)-(251,21): text "Stop"; alarm colour if .I_Btn_Stop OR .HMI_wControlWord.2; taps .I_Btn_Stop
rectangle at (150,100)-(236,131): text "Hold"; alarm colour if .HMI_wControlWord.3; toggles .HMI_wControlWord.3
rectangle at (150,130)-(236,161): text "Suspend"; alarm colour if .HMI_wControlWord.4; toggles .HMI_wControlWord.4
rectangle at (265,-10)-(466,21): text "Mode : %s"; shows .fbStateModel.eMode
rectangle at (265,20)-(466,51): text "State: %s"; shows .fbStateModel.eState
rectangle at (0,130)-(101,161): text "Manual"; alarm colour if .HMI_uModeReq=3; runs INTERN ASSIGN HMI_uModeReq:=(3)
rectangle at (0,110)-(101,131): text "Mode Selection"
rectangle at (0,160)-(101,191): text "Production1"; alarm colour if .HMI_uModeReq=5; runs INTERN ASSIGN HMI_uModeReq:=(5)
rectangle at (0,60)-(101,91): text "Covers Closed"; alarm colour if .I_CoversClosed; toggles .I_CoversClosed
rectangle at (240,100)-(326,131): text "Un-Hold"; alarm colour if .HMI_wControlWord.5; taps .HMI_wControlWord.5
rectangle at (240,130)-(326,161): text "Un-Suspend"; alarm colour if .HMI_wControlWord.6; taps .HMI_wControlWord.6
rectangle at (150,30)-(251,61): text "Complete"; alarm colour if .fbStateModel.bComplete; taps .fbStateModel.bComplete
rectangle at (150,60)-(251,91): text "ACK Completed"; alarm colour if .fbStateModel.bAck_Completed; taps .fbStateModel.bAck_Completed
ellipse at (265,50)-(316,91): text "Start"; alarm colour if .O_Light_Start
ellipse at (315,50)-(366,91): text "Stop"; alarm colour if .O_Light_Stop
ellipse at (365,50)-(416,91): text "Warning"; alarm colour if .O_Light_Warning
ellipse at (415,50)-(466,91): text "Error"; alarm colour if .O_Light_Error
rounded rectangle at (485,5)-(576,46): text "R: StopClear"; alarm colour if .O_RelayStop
rounded rectangle at (485,45)-(576,86): text "R: Emergency / StopClear"; alarm colour if .O_RelayEStop
rectangle at (0,30)-(101,61): text "E-Stop Clear"; alarm colour if .I_EStopClear; toggles .I_EStopClear
rectangle at (240,160)-(326,191): text "Continue"; alarm colour if .HMI_wControlWord.7; taps .HMI_wControlWord.7
polygon at (390,130)-(410,180): angle .fAngle1
rectangle at (350,240)-(451,261): text "Cycle: %d"; shows PRG_Production1.iCycleCount
polygon at (510,130)-(530,180): angle .fAngle2
rectangle at (0,190)-(101,221): text "Production2"; alarm colour if .HMI_uModeReq=6; runs INTERN ASSIGN HMI_uModeReq:=(6)
rectangle at (350,100)-(451,121): text "Process 1"
rectangle at (470,100)-(571,121): text "Process 2"
rectangle at (470,240)-(571,261): text "Cycle: %d"; shows PRG_Production2.iCycleCount
embedded screen at (0,270)-(581,556): VC_PackMLStates
embedded screen at (240,200)-(336,266): VC_FB_Process3
5 more shapes without text or variables
*)

(* Visualisation Visual Components/VC_FB_Process3
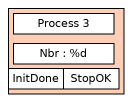
rectangle at (5,5)-(106,26): text "Process 3"
rectangle at (5,35)-(106,56): text "Nbr : %d"; shows $fb$.iProcessCount
rectangle at (0,60)-(56,81): text "InitDone"; alarm colour if $fb$.bInitDone
rectangle at (55,60)-(111,81): text "StopOK"; alarm colour if $fb$.bStopOK
1 more shapes without text or variables
*)

(* Visualisation Visual Components/VC_PackMLStates
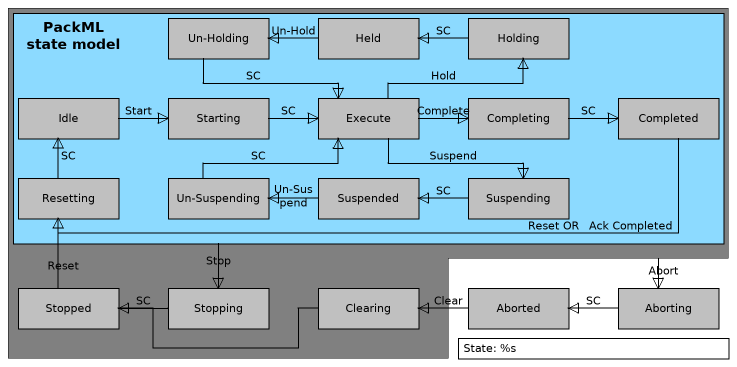
rounded rectangle at (160,280)-(261,321): text "Stopping"; alarm colour if $PackML$.eState = 4
rounded rectangle at (10,90)-(111,131): text "Idle"; alarm colour if $PackML$.eState = 6
rounded rectangle at (160,170)-(261,211): text "Un-Suspending"; alarm colour if $PackML$.eState = 11
rounded rectangle at (610,280)-(711,321): text "Aborting"; alarm colour if $PackML$.eState = 0
rounded rectangle at (460,280)-(561,321): text "Aborted"; alarm colour if $PackML$.eState = 1
rectangle at (450,330)-(721,351): text "State: %s"; shows $PackML$.strState
rounded rectangle at (310,280)-(411,321): text "Clearing"; alarm colour if $PackML$.eState = 2
rounded rectangle at (10,280)-(111,321): text "Stopped"; alarm colour if $PackML$.eState = 3
rounded rectangle at (10,170)-(111,211): text "Resetting"; alarm colour if $PackML$.eState = 5
rounded rectangle at (160,90)-(261,131): text "Starting"; alarm colour if $PackML$.eState = 7
rounded rectangle at (310,90)-(411,131): text "Execute"; alarm colour if $PackML$.eState = 8
rounded rectangle at (460,90)-(561,131): text "Completing"; alarm colour if $PackML$.eState = 15
rounded rectangle at (610,90)-(711,131): text "Completed"; alarm colour if $PackML$.eState = 16
rounded rectangle at (310,170)-(411,211): text "Suspended"; alarm colour if $PackML$.eState = 10
rounded rectangle at (460,170)-(561,211): text "Suspending"; alarm colour if $PackML$.eState = 9
rounded rectangle at (460,10)-(561,51): text "Holding"; alarm colour if $PackML$.eState = 12
rounded rectangle at (310,10)-(411,51): text "Held"; alarm colour if $PackML$.eState = 13
rounded rectangle at (160,10)-(261,51): text "Un-Holding"; alarm colour if $PackML$.eState = 14
polyline at (645,250)-(655,280): alarm colour if $PackML$.bAbort
rectangle at (635,255)-(676,271): text "Abort"; alarm colour if $PackML$.bAbort
polyline at (205,235)-(215,280): alarm colour if $PackML$.bStop
rectangle at (190,245)-(231,261): text "Stop"; alarm colour if $PackML$.bStop
polyline at (195,130)-(335,170): alarm colour if $PackML$.bSC
rectangle at (235,140)-(266,156): text "SC"; alarm colour if $PackML$.bSC
polyline at (195,50)-(335,90): alarm colour if $PackML$.bSC
polyline at (380,50)-(520,90): alarm colour if $PackML$.bHold
rectangle at (420,60)-(451,76): text "Hold"; alarm colour if $PackML$.bHold
polyline at (560,295)-(610,305): alarm colour if $PackML$.bSC
polyline at (45,210)-(55,280): alarm colour if $PackML$.bReset
polyline at (110,105)-(160,115): alarm colour if $PackML$.bStart
polyline at (110,295)-(310,340): alarm colour if $PackML$.bSC
rectangle at (230,60)-(261,76): text "SC"; alarm colour if $PackML$.bSC
polyline at (380,130)-(520,170): alarm colour if $PackML$.bSuspend
rectangle at (415,140)-(476,156): text "Suspend"; alarm colour if $PackML$.bSuspend
rectangle at (120,285)-(151,301): text "SC"; alarm colour if $PackML$.bSC
rectangle at (570,285)-(601,301): text "SC"; alarm colour if $PackML$.bSC
polyline at (410,295)-(460,305): alarm colour if $PackML$.bClear
rectangle at (420,285)-(461,301): text "Clear"; alarm colour if $PackML$.bClear
polyline at (260,105)-(310,115): alarm colour if $PackML$.bSC
rectangle at (265,95)-(296,111): text "SC"; alarm colour if $PackML$.bSC
rectangle at (110,95)-(151,111): text "Start"; alarm colour if $PackML$.bStart
rectangle at (35,250)-(76,266): text "Reset"; alarm colour if $PackML$.bReset
polyline at (410,185)-(460,195): alarm colour if $PackML$.bSC
rectangle at (420,175)-(451,191): text "SC"; alarm colour if $PackML$.bSC
polyline at (410,25)-(460,35): alarm colour if $PackML$.bSC
rectangle at (420,15)-(451,31): text "SC"; alarm colour if $PackML$.bSC
polyline at (260,185)-(310,195): alarm colour if $PackML$.bUn_Suspend
rectangle at (260,170)-(311,206): text "Un-Sus / pend"; alarm colour if $PackML$.bUn_Suspend
polyline at (260,25)-(310,35): alarm colour if $PackML$.bUn_Hold
rectangle at (260,15)-(311,31): text "Un-Hold"; alarm colour if $PackML$.bUn_Hold
polyline at (410,105)-(460,115): alarm colour if $PackML$.bComplete
rectangle at (410,95)-(461,111): text "Complete"; alarm colour if $PackML$.bComplete
polyline at (560,105)-(610,115): alarm colour if $PackML$.bSC
rectangle at (565,95)-(596,111): text "SC"; alarm colour if $PackML$.bSC
polyline at (45,130)-(55,170): alarm colour if $PackML$.bSC
rectangle at (45,140)-(76,156): text "SC"; alarm colour if $PackML$.bSC
polyline at (50,130)-(670,225): alarm colour if $PackML$.bReset OR $PackML$.Ack_Completed
rectangle at (515,210)-(576,226): text "Reset OR"; alarm colour if $PackML$.bReset
rectangle at (575,210)-(671,226): text "Ack Completed"; alarm colour if $PackML$.bAck_Completed
rectangle at (10,10)-(121,51): text "PackML / state model"
2 more shapes without text or variables
*)

(* Visualisation Visualisation items/VC_Var_Int
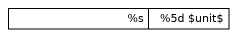
rounded rectangle at (0,0)-(141,21): text "%s"; shows $label$
rounded rectangle at (140,0)-(221,21): text "%5d $unit$"; shows $VAR$
*)

(* Visualisation Visualisation items/VC_Var_Int_edit
rounded rectangle at (0,0)-(141,21): text "%s"; shows $label$
1 elements of other kinds (tables, trends, ...) not read
*)

(* Visualisation Visualisation items/VC_Var_Real
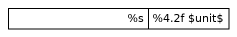
rounded rectangle at (0,0)-(141,21): text "%s"; shows $label$
rounded rectangle at (140,0)-(221,21): text "%4.2f $unit$"; shows $VAR$
*)

(* Visualisation Visualisation items/VC_Var_Real_edit
rounded rectangle at (0,0)-(141,21): text "%s"; shows $label$
1 elements of other kinds (tables, trends, ...) not read
*)
